FUNCTION_BLOCK PlantNo1
VAR_INPUT
	lrInput : LREAL := 0.0;	
END_VAR

VAR_OUTPUT
	lrOutput : LREAL := 0.0;
END_VAR

VAR
	lrLastInput : LREAL := 0.0;
	lrLastOutput : LREAL := 0.0;
	lrTs : LREAL := 0.001;
	lr2OverTs : lreal := 2/0.001;
END_VAR

lr2OverTs := 2.0 / lrTs;
lrOutput := ((lr2OverTs - 500.0) * lrLastOutput + 500.0 * (lrInput + lrLastInput)) / (lr2OverTs + 500.0);
lrLastOutput := lrOutput;
lrLastInput := lrInput;

END_FUNCTION_BLOCK

(* stored: Version 1.1.0.1, ProductVersion 3.1.4024.12
   POU PlantNo1: Id {17721785-2715-4c55-886a-12a5c9e3ba34}, SpecialFunc None *)
